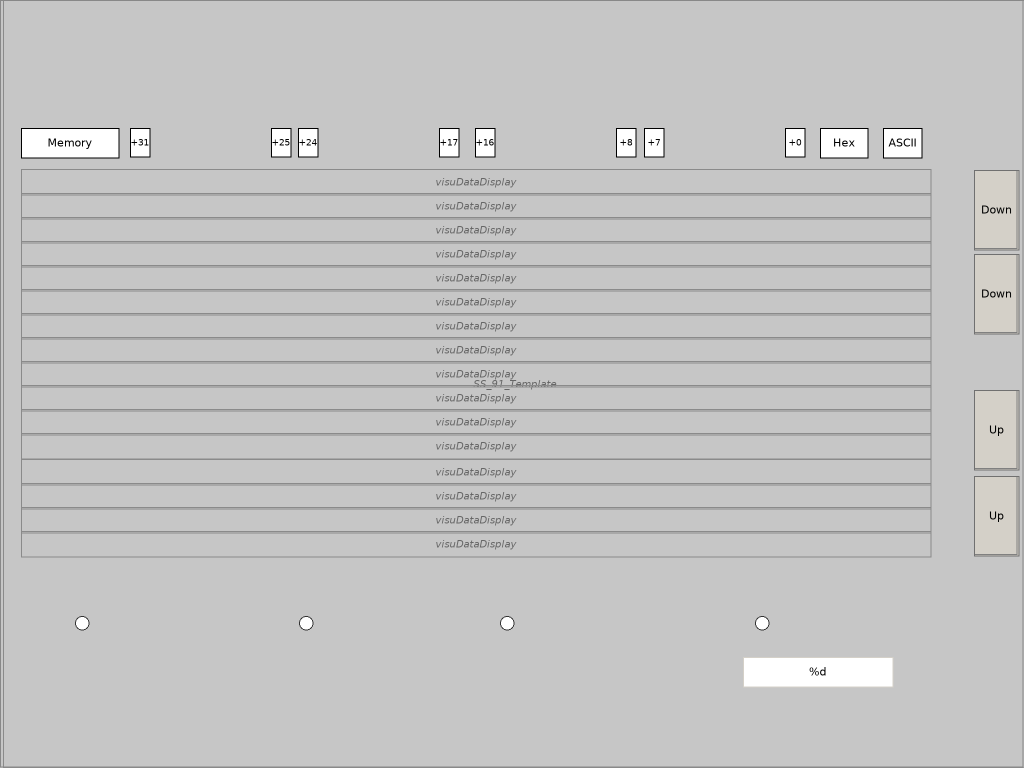
VISUALIZATION SS_80_DataDisplay  // 1024x768
    Frame (3,0 1024x768)
        shows SS_91_Template(header := gHMIData.hmiHeader)
    Frame (21,169 910x26)
        shows visuDataDisplay(d := ioview.ByteRow[0])
    Frame (21,193 910x26)
        shows visuDataDisplay(d := ioview.ByteRow[1])
    Frame (21,217 910x26)
        shows visuDataDisplay(d := ioview.ByteRow[2])
    Frame (21,241 910x26)
        shows visuDataDisplay(d := ioview.ByteRow[3])
    Frame (21,265 910x26)
        shows visuDataDisplay(d := ioview.ByteRow[4])
    Frame (21,289 910x26)
        shows visuDataDisplay(d := ioview.ByteRow[5])
    Frame (21,313 910x26)
        shows visuDataDisplay(d := ioview.ByteRow[6])
    Frame (21,337 910x26)
        shows visuDataDisplay(d := ioview.ByteRow[7])
    Frame (21,361 910x26)
        shows visuDataDisplay(d := ioview.ByteRow[8])
    Frame (21,385 910x26)
        shows visuDataDisplay(d := ioview.ByteRow[9])
    Frame (21,409 910x26)
        shows visuDataDisplay(d := ioview.ByteRow[10])
    Frame (21,433 910x26)
        shows visuDataDisplay(d := ioview.ByteRow[11])
    Rectangle (21,128 98x30), "Memory"
    Rectangle (883,128 39x30), "ASCII"
    Rectangle (820,128 48x30), "Hex"
    Rectangle (785,128 20x29), "+0"
    Rectangle (644,128 20x29), "+7"
    Rectangle (475,128 20x29), "+16"
    Rectangle (616,128 20x29), "+8"
    Rectangle (439,128 20x29), "+17"
    Rectangle (298,128 20x29), "+24"
    Rectangle (271,128 20x29), "+25"
    Rectangle (130,128 20x29), "+31"
    Frame (21,459 910x26)
        shows visuDataDisplay(d := ioview.ByteRow[12])
    Frame (21,483 910x26)
        shows visuDataDisplay(d := ioview.ByteRow[13])
    Frame (21,507 910x26)
        shows visuDataDisplay(d := ioview.ByteRow[14])
    Frame (21,531 910x26)
        shows visuDataDisplay(d := ioview.ByteRow[15])
    Button (974,476 45x80), "Up"
        tap ioView.btnRaiseFaster
    Button (974,390 45x80), "Up"
        tap ioView.btnRaise
    Button (974,254 45x80), "Down"
        tap ioView.btnLower
    Button (974,170 45x80), "Down"
        tap ioView.btnLowerFaster
    RadioButton (753,583 150x80), variable: ioView.memtype
    RadioButton (73,583 150x80), variable: ioView.memsize
    RadioButton (297,583 230x80), variable: ioView.memHexDisplay
        p340057476: HEX/DEC
    RadioButton (498,583 235x80), variable: ioView.memswap
        p2481256679: SIEMENS/754
    Textfield (743,657 150x30), "%d", text variable: ioView.memoffset
        OnMouseClick: write ioView.memoffset via VisuDialogs.Numpad
END_VISUALIZATION

(* stored: Version 1.1.0.1, ProductVersion 3.1.4024.12
   Visu SS_80_DataDisplay: Id {81d00564-ef7e-46db-b7df-86ab8833ec42} *)
